FUNCTION_BLOCK FB_Circle EXTENDS FB_Shape

METHOD Draw : STRING
ADSLOGSTR(    msgCtrlMask:=ADSLOG_MSGTYPE_LOG,
              msgFmtStr:='Drawing a %s circle',
              strArg:= SUPER^._color.applyColor());
END_METHOD

END_FUNCTION_BLOCK

(* stored: Version 1.1.0.1, ProductVersion 3.1.4024.12
   POU FB_Circle: Id {e9bbca66-4614-432d-b293-bbcc196b2130}, SpecialFunc None
   Method Draw: Id {9f53bee7-91ba-4278-9bbc-a2c57222b213} *)
